// TwinCAT 3 PLC project PLC
// ProgramVersion: 3.1.4023.0
// libraries:
//   Tc2_SerialCom, * (Beckhoff Automation GmbH)
//   Tc2_Standard, * (Beckhoff Automation GmbH)
//   Tc2_System, * (Beckhoff Automation GmbH)
//   Tc3_Module, * (Beckhoff Automation GmbH)
// project tree:
//   / Comms.TcTTO
//   GVLs/ GVL.TcGVL
//   POUs/Devices/PowerSupply/Commands/ CMD_Beep.TcPOU, CMD_LocalMode.TcPOU, CMD_RemoteMode.TcPOU, CMD_QueryTargetVoltage.TcPOU
//   POUs/Devices/PowerSupply/ PowerSupply.TcPOU
//   POUs/Devices/SerialPort/ SerialPort.TcPOU
//   POUs/Lib/CommandBuffer/ CommandBuffer.TcPOU
//   POUs/Lib/Commands/ CommandNull.TcPOU, I_Command.TcIO
//   POUs/Lib/ComPort/ ComPort.TcPOU
//   POUs/Lib/Interfaces/ I_CommsReceiver.TcIO, I_CommsTransceiver.TcIO, I_CommsTransmitter.TcIO
//   POUs/Lib/WatchDog/ WatchDog.TcPOU
//   POUs/ MAIN.TcPOU
// real-time tasks:
//   TASK Comms: cycle T#1ms, priority 1, ADS port 351
// I/O:
//   DEVICE Device 1 (EtherCAT), AmsNetId 5.59.22.14.6.1
//     Term 1 (EK1100) [EK1100 EtherCAT Coupler (2A E-Bus)]
//       Term 2 (EL6002) [EL6002 Interface 2Ch. (RS232)]

CONFIGURATION PLC
    RESOURCE PLC ON TwinCAT3
        TASK Comms(INTERVAL := T#1ms, PRIORITY := 1);
        PROGRAM MAIN WITH Comms : MAIN;
    END_RESOURCE
END_CONFIGURATION

// ---- GVLs/GVL.TcGVL
VAR_GLOBAL

	serialPort1 : SerialPort;
	powerSupply : PowerSupply(serialPort1);
	
END_VAR

// ---- POUs/Lib/Commands/I_Command.TcIO
INTERFACE I_Command

METHOD Destroy
VAR_INPUT
END_VAR
END_METHOD

METHOD PUBLIC Execute : BOOL
VAR_INPUT
END_VAR
END_METHOD

PROPERTY PUBLIC isBusy : BOOL
GET
END_GET
END_PROPERTY

PROPERTY isComplete : BOOL
GET
END_GET
END_PROPERTY

END_INTERFACE

// ---- POUs/Lib/Interfaces/I_CommsReceiver.TcIO
INTERFACE I_CommsReceiver

METHOD PUBLIC ConfigureRead
VAR_INPUT
	Prefix: STRING;
	Suffix: STRING;
	Timeout: TIME;
END_VAR
END_METHOD

{attribute 'monitoring' := 'call'}
PROPERTY PUBLIC hasReceivedData : BOOL
GET
END_GET
END_PROPERTY

METHOD PUBLIC Read : String
VAR_INPUT
END_VAR
END_METHOD

END_INTERFACE

// ---- POUs/Lib/Interfaces/I_CommsTransceiver.TcIO
INTERFACE I_CommsTransceiver EXTENDS I_CommsReceiver, I_CommsTransmitter

END_INTERFACE

// ---- POUs/Lib/Interfaces/I_CommsTransmitter.TcIO
INTERFACE I_CommsTransmitter

{attribute 'monitoring' := 'call'}
PROPERTY hasError : BOOL
GET
END_GET
END_PROPERTY

{attribute 'monitoring' := 'call'}
PROPERTY isBusy : BOOL
GET
END_GET
END_PROPERTY

METHOD PUBLIC Send
VAR_INPUT
	str : STRING;
END_VAR
END_METHOD

END_INTERFACE

// ---- POUs/MAIN.TcPOU
PROGRAM MAIN
VAR
	connect: BOOL;
	disconnect: BOOL;
	beep: BOOL;
	queryTargetVoltage: BOOL;
	targetVoltage : LREAL;
END_VAR

serialPort1.CyclicCall();
powerSupply.CyclicCall();

// control of the PSU
IF connect THEN
	connect := FALSE;
	powerSupply.Connect();
END_IF

IF disconnect THEN
	disconnect := FALSE;
	powerSupply.Disconnect();
END_IF

IF beep THEN
	beep := FALSE;
	powerSupply.Beep();
END_IF

IF queryTargetVoltage THEN
	queryTargetVoltage := FALSE;
	powerSupply.QueryTargetVoltage();
END_IF

targetVoltage := powerSupply.TargetVoltage;

END_PROGRAM

// ---- POUs/Devices/PowerSupply/PowerSupply.TcPOU
FUNCTION_BLOCK PowerSupply
VAR
	ComHandler : I_CommsTransceiver;
	CommandBuffer : CommandBuffer;
	_targetVoltage : LREAL;
END_VAR

METHOD PUBLIC Beep
VAR
	newCommand : POINTER TO CMD_Beep;
END_VAR
IF NOT CommandBuffer.isFull THEN 
	newCommand := __NEW(CMD_Beep(Comms := THIS^.ComHandler));
	CommandBuffer.Insert(newCommand^); 
END_IF
END_METHOD

METHOD PUBLIC Connect
VAR
	newCommand: POINTER TO CMD_RemoteMode;
END_VAR
IF NOT CommandBuffer.isFull THEN 
	newCommand := __NEW(CMD_RemoteMode(Comms := THIS^.ComHandler));
	CommandBuffer.Insert(newCommand^); 
END_IF
END_METHOD

METHOD PUBLIC CyclicCall
CommandBuffer.CurrentCommand.Execute();
		
IF CommandBuffer.CurrentCommand.isComplete THEN 
	CommandBuffer.Next();
	RETURN;
END_IF
END_METHOD

METHOD PUBLIC Disconnect
VAR
	newCommand: POINTER TO CMD_LocalMode;
END_VAR
IF NOT CommandBuffer.isFull THEN 
	newCommand := __NEW(CMD_LocalMode(Comms := THIS^.ComHandler));
	CommandBuffer.Insert(newCommand^); 
END_IF
END_METHOD

METHOD FB_init : BOOL
VAR_INPUT
	bInitRetains : BOOL; // if TRUE, the retain variables are initialized (warm start / cold start)
	bInCopyCode : BOOL;  // if TRUE, the instance afterwards gets moved into the copy code (online change)
	Comms : I_CommsTransceiver;
END_VAR
THIS^.ComHandler := Comms;
END_METHOD

METHOD PUBLIC QueryTargetVoltage
VAR
	newCommand: POINTER TO CMD_QueryTargetVoltage;
END_VAR
IF NOT CommandBuffer.isFull THEN 
	newCommand := __NEW(CMD_QueryTargetVoltage(Comms := THIS^.ComHandler, ReferenceToResult:=_targetVoltage));
	CommandBuffer.Insert(newCommand^); 
END_IF
END_METHOD

PROPERTY PUBLIC TargetVoltage : LREAL
GET
TargetVoltage := this^._targetVoltage;
END_GET
END_PROPERTY

END_FUNCTION_BLOCK

// ---- POUs/Lib/CommandBuffer/CommandBuffer.TcPOU
FUNCTION_BLOCK CommandBuffer
VAR_INPUT
END_VAR
VAR_OUTPUT
END_VAR
VAR
	commandArray : ARRAY [0..MAX_ENTRIES] OF I_Command;
	lastIndex : INT := EMPTY;
	emptyCommand : CommandNull;
END_VAR
VAR CONSTANT
	EMPTY : INT := -1;
	MAX_ENTRIES : INT := 10;
	FIRST_ENTRY : INT := 0;
	LAST_ENTRY : INT := MAX_ENTRIES -1;
END_VAR

PROPERTY PUBLIC CurrentCommand : I_Command
GET
IF isEmpty THEN
	CurrentCommand := emptyCommand;
ELSE 
	CurrentCommand := commandArray[FIRST_ENTRY];
END_IF
END_GET
END_PROPERTY

METHOD PUBLIC Insert : BOOL
VAR_INPUT
	cmd : I_Command;
END_VAR
IF isFull THEN
	RETURN;
END_IF

lastIndex := lastIndex + 1;
commandArray[lastIndex] := cmd;
Insert := TRUE;
END_METHOD

PROPERTY PUBLIC isEmpty : BOOL
GET
isEmpty := (lastIndex = EMPTY);
END_GET
END_PROPERTY

PROPERTY PUBLIC isFull : BOOL
GET
isFull := (lastIndex = MAX_ENTRIES);
END_GET
END_PROPERTY

METHOD PUBLIC Next
VAR_INPUT
END_VAR
IF isEmpty THEN
	RETURN;
END_IF

Shift();
END_METHOD

METHOD PRIVATE Shift
VAR_INPUT
END_VAR
VAR
	i: INT;
END_VAR
commandArray[FIRST_ENTRY].Destroy();

FOR i := 1 TO lastIndex + 1 DO
	commandArray[i-1] := commandArray[i];
END_FOR

lastIndex := lastIndex - 1;
END_METHOD

END_FUNCTION_BLOCK

// ---- POUs/Lib/Commands/CommandNull.TcPOU
{attribute 'enable_dynamic_creation'}
FUNCTION_BLOCK CommandNull IMPLEMENTS I_Command
VAR_INPUT
END_VAR
VAR_OUTPUT
END_VAR

METHOD Destroy
VAR_INPUT
END_VAR
END_METHOD

METHOD PUBLIC Execute : BOOL
VAR_INPUT
END_VAR
END_METHOD

PROPERTY PUBLIC hasTimedOut : BOOL
GET
hasTimedOut := false;
END_GET
END_PROPERTY

PROPERTY PUBLIC isBusy : BOOL
GET
isBusy := false;
END_GET
END_PROPERTY

PROPERTY isComplete : BOOL
GET
isComplete := true;
END_GET
END_PROPERTY

END_FUNCTION_BLOCK

// ---- POUs/Devices/PowerSupply/Commands/CMD_Beep.TcPOU
{attribute 'enable_dynamic_creation'}
FUNCTION_BLOCK CMD_Beep IMPLEMENTS I_Command
VAR_INPUT
END_VAR
VAR_OUTPUT
END_VAR
VAR
	Comms : I_CommsTransmitter;
	Status : (IDLE, EXECUTE, SENDING, SENT, COMPLETE, TIMED_OUT);
	WatchDog : WatchDog; 
END_VAR
VAR CONSTANT
	CMD : STRING := 'SYSTem:BEEPer$R$N';
	TIME_OUT : TIME := T#2S;	
END_VAR

CASE Status OF
	
	EXECUTE: 
		WatchDog.Enable(TIME_OUT);
		Status := SENDING;
		
	SENDING:
		IF Comms.isBusy THEN
			RETURN;
		ELSE
			Comms.Send(CMD);
			Status := SENT;
		END_IF
		
	SENT:
		IF Comms.isBusy THEN
			RETURN;
		ELSE
			WatchDog.Disable();
			Status := COMPLETE;
		END_IF
		
	IDLE: //
	COMPLETE://
	TIMED_OUT: //
	
END_CASE

IF WatchDog.isTriggered THEN
	WatchDog.Disable();
	Status := TIMED_OUT;
END_IF

METHOD Destroy
VAR_INPUT
END_VAR
VAR
	selfPointer: POINTER TO CMD_Beep;
END_VAR
selfPointer := ADR(THIS^);
__DELETE(selfPointer);
END_METHOD

METHOD PUBLIC Execute : BOOL
VAR_INPUT

END_VAR
IF NOT isBusy THEN
	Status := EXECUTE;
	Execute := TRUE;
END_IF

THIS^();
END_METHOD

METHOD FB_init : BOOL
VAR_INPUT
	bInitRetains : BOOL; // if TRUE, the retain variables are initialized (warm start / cold start)
	bInCopyCode : BOOL;  // if TRUE, the instance afterwards gets moved into the copy code (online change)
	Comms : I_CommsTransmitter;
END_VAR
THIS^.Comms := Comms;
END_METHOD

PROPERTY PUBLIC hasTimedOut : BOOL
GET
hasTimedOut := (Status = TIMED_OUT) ;
END_GET
END_PROPERTY

PROPERTY PUBLIC isBusy : BOOL
GET
isBusy := not (Status = IDLE or Status = COMPLETE or Status = TIMED_OUT);
END_GET
END_PROPERTY

PROPERTY isComplete : BOOL
GET
isComplete := (Status = COMPLETE or Status = TIMED_OUT) ;
END_GET
END_PROPERTY

END_FUNCTION_BLOCK

// ---- POUs/Lib/WatchDog/WatchDog.TcPOU
FUNCTION_BLOCK WatchDog
VAR_INPUT
END_VAR
VAR_OUTPUT
END_VAR
VAR
	Timer : TON;
	Enabled : BOOL;
	TimeSpan : TIME := T#1S;
END_VAR

Timer(IN:=Enabled, PT:=TimeSpan);

METHOD PUBLIC Disable : BOOL
VAR_INPUT
END_VAR
Enabled := FALSE;
THIS^();
END_METHOD

METHOD PUBLIC Enable
VAR_INPUT
	Duration : TIME;
END_VAR
TimeSpan := Duration;
Enabled := TRUE;
THIS^();
END_METHOD

PROPERTY PUBLIC isTriggered : BOOL
GET
THIS^();
isTriggered := Timer.Q;
END_GET
END_PROPERTY

METHOD PUBLIC Reset : BOOL
VAR_INPUT
END_VAR
Disable();
Enable(TimeSpan);
END_METHOD

END_FUNCTION_BLOCK

// ---- POUs/Devices/PowerSupply/Commands/CMD_RemoteMode.TcPOU
{attribute 'enable_dynamic_creation'}
FUNCTION_BLOCK CMD_RemoteMode IMPLEMENTS I_Command
VAR_INPUT
END_VAR
VAR_OUTPUT
END_VAR
VAR
	Comms : I_CommsTransmitter;
	Status : (IDLE, EXECUTE, SENDING, SENT, COMPLETE, TIMED_OUT);
	WatchDog : WatchDog; 
END_VAR
VAR CONSTANT
	CMD : STRING := 'SYSTem:REMote$R$N';
	TIME_OUT : TIME := T#2S;	
END_VAR

CASE Status OF
	
	EXECUTE: 
		WatchDog.Enable(TIME_OUT);
		Status := SENDING;
		
	SENDING:
		IF Comms.isBusy THEN
			RETURN;
		ELSE
			Comms.Send(CMD);
			Status := SENT;
		END_IF
		
	SENT:
		IF Comms.isBusy THEN
			RETURN;
		ELSE
			WatchDog.Disable();
			Status := COMPLETE;
		END_IF

	IDLE: //
	COMPLETE://
	TIMED_OUT: //
	
END_CASE

IF WatchDog.isTriggered THEN
	WatchDog.Disable();
	Status := TIMED_OUT;
END_IF

METHOD Destroy
VAR_INPUT
END_VAR
VAR
	selfPointer: POINTER TO CMD_RemoteMode;
END_VAR
selfPointer := ADR(THIS^);
__DELETE(selfPointer);
END_METHOD

METHOD PUBLIC Execute : BOOL
VAR_INPUT
END_VAR
IF NOT isBusy THEN
	Status := EXECUTE;
	Execute := TRUE;
END_IF

THIS^();
END_METHOD

METHOD FB_init : BOOL
VAR_INPUT
	bInitRetains : BOOL; // if TRUE, the retain variables are initialized (warm start / cold start)
	bInCopyCode : BOOL;  // if TRUE, the instance afterwards gets moved into the copy code (online change)
	Comms : I_CommsTransmitter;
END_VAR
THIS^.Comms := Comms;
END_METHOD

PROPERTY PUBLIC hasTimedOut : BOOL
GET
hasTimedOut := (Status = TIMED_OUT) ;
END_GET
END_PROPERTY

PROPERTY PUBLIC isBusy : BOOL
GET
isBusy := not (Status = IDLE or Status = COMPLETE or Status = TIMED_OUT);
END_GET
END_PROPERTY

PROPERTY isComplete : BOOL
GET
isComplete := (Status = COMPLETE or Status = TIMED_OUT) ;
END_GET
END_PROPERTY

END_FUNCTION_BLOCK

// ---- POUs/Devices/PowerSupply/Commands/CMD_LocalMode.TcPOU
{attribute 'enable_dynamic_creation'}
FUNCTION_BLOCK CMD_LocalMode IMPLEMENTS I_Command
VAR_INPUT
END_VAR
VAR_OUTPUT
END_VAR
VAR
	Comms : I_CommsTransmitter;
	Status : (IDLE, EXECUTE, SENDING, SENT, COMPLETE, TIMED_OUT);
	WatchDog : WatchDog; 
END_VAR
VAR CONSTANT
	CMD : STRING := 'SYSTem:LOCal$R$N';
	TIME_OUT : TIME := T#2S;	
END_VAR

CASE Status OF
	
	EXECUTE: 
		WatchDog.Enable(TIME_OUT);
		Status := SENDING;
		
	SENDING:
		IF Comms.isBusy THEN
			RETURN;
		ELSE
			Comms.Send(CMD);
			Status := SENT;
		END_IF
		
	SENT:
		IF Comms.isBusy THEN
			RETURN;
		ELSE
			WatchDog.Disable();
			Status := COMPLETE;
		END_IF

	IDLE: //
	COMPLETE://
	TIMED_OUT: //
	
END_CASE

IF WatchDog.isTriggered THEN
	WatchDog.Disable();
	Status := TIMED_OUT;
END_IF

METHOD Destroy
VAR_INPUT
END_VAR
VAR
	selfPointer: POINTER TO CMD_LocalMode;
END_VAR
selfPointer := ADR(THIS^);
__DELETE(selfPointer);
END_METHOD

METHOD PUBLIC Execute : BOOL
VAR_INPUT
END_VAR
IF NOT isBusy THEN
	Status := EXECUTE;
	Execute := TRUE;
END_IF

THIS^();
END_METHOD

METHOD FB_init : BOOL
VAR_INPUT
	bInitRetains : BOOL; // if TRUE, the retain variables are initialized (warm start / cold start)
	bInCopyCode : BOOL;  // if TRUE, the instance afterwards gets moved into the copy code (online change)
	Comms : I_CommsTransmitter;
END_VAR
THIS^.Comms := Comms;
END_METHOD

PROPERTY PUBLIC hasTimedOut : BOOL
GET
hasTimedOut := (Status = TIMED_OUT) ;
END_GET
END_PROPERTY

PROPERTY PUBLIC isBusy : BOOL
GET
isBusy := not (Status = IDLE or Status = COMPLETE or Status = TIMED_OUT);
END_GET
END_PROPERTY

PROPERTY isComplete : BOOL
GET
isComplete := (Status = COMPLETE or Status = TIMED_OUT) ;
END_GET
END_PROPERTY

END_FUNCTION_BLOCK

// ---- POUs/Devices/PowerSupply/Commands/CMD_QueryTargetVoltage.TcPOU
{attribute 'enable_dynamic_creation'}
FUNCTION_BLOCK CMD_QueryTargetVoltage IMPLEMENTS I_Command
VAR_INPUT
END_VAR
VAR_OUTPUT
END_VAR
VAR
	Comms : I_CommsTransceiver;
	Status : (IDLE, EXECUTE, CONFIG_RECEIVER, SENDING_QUERY, SENT_QUERY, WAITING_FOR_REPLY, PROCESSING_REPLY, COMPLETE, TIMED_OUT);
	WatchDog : WatchDog; 
	
	receivedString : STRING;
	result : REFERENCE TO LREAL;
	
END_VAR
VAR CONSTANT
	CMD : STRING := 'SOUR:VOLT:AMPL?$R$N';
	TIME_OUT : TIME := T#2S;	
END_VAR

CASE Status OF
	
	EXECUTE: 
		WatchDog.Enable(TIME_OUT);
		Status := CONFIG_RECEIVER;
		
	CONFIG_RECEIVER:
		Comms.ConfigureRead(Prefix:='',Suffix:='$R$N',Timeout:=TIME_OUT);
		Status := SENDING_QUERY;
		
	SENDING_QUERY:
		IF Comms.isBusy THEN
			RETURN;
		ELSE
			Comms.Send(CMD);
			Status := SENT_QUERY;
		END_IF
		
	SENT_QUERY:
		IF Comms.isBusy THEN
			RETURN;
		ELSE
			WatchDog.Disable();
			Status := WAITING_FOR_REPLY;
		END_IF
		
	WAITING_FOR_REPLY:
		IF Comms.hasReceivedData THEN
			receivedString := Comms.Read();
			Status := PROCESSING_REPLY;
		END_IF
		
	PROCESSING_REPLY:
		result := ConvertTargetVoltageStringToReal(receivedString);
		Status := COMPLETE;
		
	IDLE: //
	COMPLETE://
	TIMED_OUT: //
	
END_CASE

IF WatchDog.isTriggered THEN
	WatchDog.Disable();
	Status := TIMED_OUT;
END_IF

METHOD PRIVATE ConvertTargetVoltageStringToReal : lreal
VAR_INPUT
	encodedString : STRING;
END_VAR
ConvertTargetVoltageStringToReal := STRING_TO_LREAL(encodedString);
END_METHOD

METHOD Destroy
VAR_INPUT
END_VAR
VAR
	selfPointer: POINTER TO CMD_Beep;
END_VAR
selfPointer := ADR(THIS^);
__DELETE(selfPointer);
END_METHOD

METHOD PUBLIC Execute : BOOL
VAR_INPUT

END_VAR
IF NOT isBusy THEN
	Status := EXECUTE;
	Execute := TRUE;
END_IF

THIS^();
END_METHOD

METHOD FB_init : BOOL
VAR_INPUT
	bInitRetains : BOOL; // if TRUE, the retain variables are initialized (warm start / cold start)
	bInCopyCode : BOOL;  // if TRUE, the instance afterwards gets moved into the copy code (online change)
	Comms : I_CommsTransceiver;
	ReferenceToResult : REFERENCE TO LREAL;
END_VAR
THIS^.Comms := Comms;
THIS^.result REF= ReferenceToResult;
END_METHOD

PROPERTY PUBLIC hasTimedOut : BOOL
GET
hasTimedOut := (Status = TIMED_OUT) ;
END_GET
END_PROPERTY

PROPERTY PUBLIC isBusy : BOOL
GET
isBusy := not (Status = IDLE or Status = COMPLETE or Status = TIMED_OUT);
END_GET
END_PROPERTY

PROPERTY isComplete : BOOL
GET
isComplete := (Status = COMPLETE or Status = TIMED_OUT) ;
END_GET
END_PROPERTY

END_FUNCTION_BLOCK

// ---- POUs/Devices/SerialPort/SerialPort.TcPOU
FUNCTION_BLOCK SerialPort IMPLEMENTS I_CommsTransceiver
VAR
	ComPort : ComPort;
	fbSendString : SendString;
	txBuffer : REFERENCE TO ComBuffer;
	txError	: BOOL;
	txErrorId: ComError_t;
	txBusy : BOOL;
	txString : STRING;
	fbReceiveString : ReceiveString;
	rxBuffer : REFERENCE TO ComBuffer;
	rxPrefix : STRING;
	rxSuffex : STRING;
	rxError	: BOOL;
	rxErrorId: ComError_t;
	rxWatchdogTime : TIME;
	rxTimeOut : BOOL;
	rxBusy : BOOL;
	rxString : STRING;
	rxCounter : INT;
END_VAR

METHOD PRIVATE CompleteRead
VAR_INPUT
END_VAR
rxString := '';
END_METHOD

{attribute 'TcRpcEnable'}
METHOD PUBLIC ConfigureRead
VAR_INPUT
	Prefix: STRING;
	Suffix: STRING;
	Timeout: TIME;
END_VAR
rxPrefix := Prefix;
rxSuffex := Suffix;
rxWatchdogTime := Timeout;
END_METHOD

METHOD PUBLIC CyclicCall
VAR_INPUT
END_VAR
ComPort();
ProcessSendData();
ProcessReceiveData();
END_METHOD

{attribute 'monitoring' := 'call'}
PROPERTY PUBLIC ErrorId : ComError_t
GET
ErrorId := txErrorId;
END_GET
END_PROPERTY

METHOD FB_init : BOOL
VAR_INPUT
	bInitRetains : BOOL; // if TRUE, the retain variables are initialized (warm start / cold start)
	bInCopyCode : BOOL;  // if TRUE, the instance afterwards gets moved into the copy code (online change)
END_VAR
txBuffer REF= THIS^.ComPort.TxBuffer;
rxBuffer REF= THIS^.ComPort.RxBuffer;
END_METHOD

{attribute 'monitoring' := 'call'}
PROPERTY PUBLIC hasError : BOOL
GET
hasError := txError;
END_GET
END_PROPERTY

{attribute 'monitoring' := 'call'}
PROPERTY PUBLIC hasReceivedData : BOOL
GET
hasReceivedData := rxString <> '';
END_GET
END_PROPERTY

{attribute 'monitoring' := 'call'}
PROPERTY PUBLIC isBusy : BOOL
GET
isBusy := txBusy;
END_GET
END_PROPERTY

METHOD PRIVATE ProcessReceiveData
VAR_INPUT
END_VAR
VAR
	sReceivedString : STRING;
END_VAR
fbReceiveString(
	Prefix:= rxPrefix,
	Suffix:= rxSuffex,
	Timeout:= rxWatchdogTime,
	ReceivedString:= sReceivedString,
	RXbuffer:= rxBuffer,
	StringReceived=> ,
	Busy=> rxBusy,
	Error=> ,
	RxTimeout=> rxTimeOut );
IF fbReceiveString.Error <> COMERROR_NOERROR THEN
	rxError := TRUE;
	rxErrorId := fbReceiveString.Error;
END_IF
IF fbReceiveString.StringReceived THEN
	rxString := sReceivedString;
	rxCounter := rxCounter + 1;
END_IF
END_METHOD

METHOD PRIVATE ProcessSendData
VAR_INPUT
END_VAR
IF txString <> '' OR fbSendString.Busy THEN
	fbSendString(	SendString:= txString,
			TXbuffer := txBuffer,
			Busy=> txBusy,
			Error=> );
	IF fbSendString.Error <> COMERROR_NOERROR THEN
		txError := TRUE;
		txErrorId := fbSendString.Error;
	END_IF
	IF fbSendString.Busy = FALSE THEN
		txString := '';
	END_IF
END_IF
END_METHOD

{attribute 'TcRpcEnable'}
METHOD PUBLIC Read : String
VAR_INPUT
END_VAR
Read := rxString;
CompleteRead();
END_METHOD

{attribute 'TcRpcEnable'}
METHOD PUBLIC Reset
VAR_INPUT
END_VAR
ComPort.Reset();

txError := FALSE;
txErrorId := COMERROR_NOERROR;

txString := '';
END_METHOD

{attribute 'TcRpcEnable'}
METHOD PUBLIC Send
VAR_INPUT
	str : STRING;
END_VAR
IF isBusy THEN 
	RETURN;
END_IF

IF str <> '' THEN
	txString := str;
	THIS^.ProcessSendData();
END_IF
END_METHOD

END_FUNCTION_BLOCK

// ---- POUs/Lib/ComPort/ComPort.TcPOU
FUNCTION_BLOCK ComPort
VAR_INPUT
END_VAR
VAR_OUTPUT
END_VAR
VAR
	(* 	I/O variables for a EL6001 terminal*)
	{attribute 'OPC.UA.DA' := '0'}
	stIn_EL6001 AT %I* : EL6inData22B;	(* linked to the EL6001 in the TwinCAT System Manager *)
	{attribute 'OPC.UA.DA' := '0'}
	stOut_EL6001 AT %Q*	: EL6outData22B;(* linked to the EL6001 in the TwinCAT System Manager *)
	
	(* Internal Variables *) 
	{attribute 'OPC.UA.DA' := '0'}
	fbComPortCtrl : SerialLineControl;
	{attribute 'OPC.UA.DA' := '0'}
	aRxBuffer : ComBuffer;
	{attribute 'OPC.UA.DA' := '0'}
	aTxBuffer : ComBuffer;
	{attribute 'OPC.UA.DA' := '0'}
	bComPortError : BOOL;
	{attribute 'OPC.UA.DA' := '0'}
	eComPortErrorId : ComError_t;

END_VAR

fbComPortCtrl(
	Mode:= SERIALLINEMODE_EL6_22B, 
	pComIn:= ADR(stIn_EL6001), 
	pComOut:= ADR(stOut_EL6001), 
	SizeComIn:= SIZEOF(stIn_EL6001), 
	Error=> , 
	ErrorID=> , 
	TxBuffer:= aTxBuffer, 
	RxBuffer:= aRxBuffer );
IF fbComPortCtrl.Error THEN
	bComPortError := TRUE;
	eComPortErrorId := fbComPortCtrl.ErrorID;
END_IF

PROPERTY PUBLIC ComPortError : BOOL
GET
ComPortError := bComPortError;
END_GET
END_PROPERTY

PROPERTY PUBLIC ComPortErrorId : ComError_t
GET
ComPortErrorId := eComPortErrorId;
END_GET
END_PROPERTY

METHOD PUBLIC Reset
VAR_INPUT
END_VAR
bComPortError := FALSE;
eComPortErrorId := COMERROR_NOERROR;
END_METHOD

PROPERTY PUBLIC RxBuffer : Reference to ComBuffer
GET
RxBuffer REF= aRxBuffer;
END_GET
END_PROPERTY

PROPERTY PUBLIC TxBuffer : Reference to ComBuffer
GET
TxBuffer REF= aTxBuffer;
END_GET
END_PROPERTY

END_FUNCTION_BLOCK
